(* IEC 61131-3 sources: POMIRTS_lab3/AS/Library/DPMaster, 3 files *)

(* ---- DPMaster.typ ---- *)
(********************************************************************
 * COPYRIGHT -- Bernecker + Rainer
 ********************************************************************
 * Library: DPMaster
 * File: DPMaster.typ
 * Author: B+R
 ********************************************************************
 * Data types of library DPMaster
 ********************************************************************)

TYPE
	DPDevice_typ : STRUCT			(*internal use*)
		DevType	: USINT ;
		MemorySize	: USINT ;
		DevAdress	: UDINT ;
		DevInfo	: UDINT ;
		DPIdent	: UDINT ;
		DevNumber	: UINT ;
		ConfMsgNr	: USINT ;
		CommandMsgNr	: USINT ;
		StatusMsgNr	: USINT ;
		OtherMsgNr	: USINT ;
	END_STRUCT;
END_TYPE

(* ---- DPMaster.fun ---- *)
(********************************************************************
 * COPYRIGHT -- Bernecker + Rainer
 ********************************************************************
 * Library: DPMaster
 * File: DPMaster.fun
 * Author: B+R
 ********************************************************************
 * Functions and function blocks of library DPMaster
 ********************************************************************)

FUNCTION_BLOCK DPMInit                 (*searches and initializes the specified device*)
	VAR_INPUT
		enable	:BOOL;                 (*enables execution*)
		Device	:UDINT;                (*device name given as pointer, e.g., "SL2.SS1.IF1"*)
	END_VAR
	VAR_OUTPUT
		status	:UINT;                 (*execution status: ERR_OK, ERR_FUB_ENABLE_FALSE, 0xXXXX = see help*)
		MemSize	:USINT;                (*indicates the DPM size on the card.*)
		DevIdent	:UDINT;            (*device identifier*)
		Run	:BOOL;                     (*device in run: TRUE = in run, FALSE = not in run*)
		Configuration	:BOOL;         (*configuration: TRUE = valid, FALSE = not valid*)
	END_VAR
END_FUNCTION_BLOCK

FUNCTION_BLOCK DPMio                   (*copies the input and output data areas between the B&R card and the specified buffers; asynchronous execution*)
	VAR_INPUT
		enable	:BOOL;                 (*enables execution*)
		DevIdent	:UDINT;            (*device identifier returned from DPMInit*)
		OutBuffer	:UDINT;            (*pointer to the output data area*)
		OutLen	:UDINT;                (*length of the output data area*)
		InBuffer	:UDINT;            (*pointer to the input data area*)
		InLen	:UDINT;                (*length of the input data area*)
	END_VAR
	VAR_OUTPUT
		status	:UINT;                 (*execution status: ERR_OK, ERR_FUB_ENABLE_FALSE, ERR_FUB_BUSY, 0xXXXX = see help*)
	END_VAR
	VAR
		hmode	:USINT;                (*internal variable*)
	END_VAR
END_FUNCTION_BLOCK

FUNCTION_BLOCK DPMStop                 (*stops the I/O exchange process*)
	VAR_INPUT
		enable	:BOOL;                 (*enables execution*)
		DevIdent	:UDINT;            (*device identifier returned from DPMInit*)
	END_VAR
	VAR_OUTPUT
		status	:UINT;                 (*execution status: ERR_OK, ERR_FUB_ENABLE_FALSE, 0xXXXX = see help*)
	END_VAR
END_FUNCTION_BLOCK

FUNCTION_BLOCK DPMCommand              (*Sends commands directly to bus stations; asynchronous execution*)
	VAR_INPUT
		enable	:BOOL;                 (*enables execution*)
		DevIdent	:UDINT;            (*device identifier returned from DPMInit*)
		RemoteAdress	:USINT;        (*remote slave node number, 1..126 = slave with specified node number, 127 = broadcast to all slaves*)
		GroupSelect	:USINT;            (*selects the slave group, 0 = only remoteAdress applies, 1..255 = slaves in specified goup*)
		Command	:USINT;                (*spezifies the type of command, e.g., freeze*)
	END_VAR
	VAR_OUTPUT
		status	:UINT;                 (*execution status: ERR_OK, ERR_FUB_ENABLE_FALSE, ERR_FUB_BUSY, 0xXXXX = see help*)
	END_VAR
	VAR
		istate	:UDINT;                (*internal variable*)
		waitCnt	:UINT;                 (*internal variable*)
		MessageHeader1	:USINT;        (*internal variable*)
		MessageHeader2	:USINT;        (*internal variable*)
		MessageHeader3	:USINT;        (*internal variable*)
		MessageHeader4	:USINT;        (*internal variable*)
		MessageHeader5	:USINT;        (*internal variable*)
		MessageHeader6	:USINT;        (*internal variable*)
		MessageHeader7	:USINT;        (*internal variable*)
		MessageHeader8	:USINT;        (*internal variable*)
	END_VAR
END_FUNCTION_BLOCK

FUNCTION_BLOCK DPMConfig               (*downloads the configuration; asynchronous execution*)
	VAR_INPUT
		enable	:BOOL;                 (*enables execution*)
		DevIdent	:UDINT;            (*device identifier returned from DPMInit*)
		ConfModulName	:UDINT;        (*configuration module name given as pointer*)
		Mode	:BOOL;                 (*download mode, TRUE = sequential, FALSE = in one step*)
	END_VAR
	VAR_OUTPUT
		status	:UINT;                 (*execution status: ERR_OK, ERR_FUB_ENABLE_FALSE, ERR_FUB_BUSY, 0xXXXX = see help*)
		Remaining	:UDINT;            (*displays the remaining segments until the configuration is completely loaded*)
	END_VAR
	VAR
		istate	:UDINT;                (*internal variable*)
		FileLength	:UINT;             (*internal variable*)
		waitCnt	:UINT;                 (*internal variable*)
		OffsetCopy	:UDINT;            (*internal variable*)
		pData	:UDINT;                (*internal variable*)
		Ready	:USINT;                (*internal variable*)
		FirstMessage	:BOOL;         (*internal variable*)
		MsgPutReady	:BOOL;             (*internal variable*)
	END_VAR
END_FUNCTION_BLOCK

FUNCTION_BLOCK DPMSlaveStat            (*returns the current slave status*)
	VAR_INPUT
		enable	:BOOL;                 (*enables execution*)
		DevIdent	:UDINT;            (*device identifier returned from DPMInit*)
		SlaveReady	:UDINT;            (*pointer to a 16 byte array indicating whether a slave is in data transfer mode*)
		SlaveDiag	:UDINT;            (*pointer to a 16 byte array indicating availability of diagnose information on slaves*)
	END_VAR
	VAR_OUTPUT
		status	:UINT;                 (*execution status: ERR_OK, ERR_FUB_ENABLE_FALSE, 0xXXXX = see help*)
		SlaveStatus	:BOOL;             (*TRUE = a configured slave is not in data transfer mode or has diagnostic messages*)
	END_VAR
END_FUNCTION_BLOCK

FUNCTION_BLOCK DPMSlaveExtStat         (*returns the exact status of a slave; asynchronous execution*)
	VAR_INPUT
		enable	:BOOL;                 (*enables execution*)
		DevIdent	:UDINT;            (*device identifier returned from DPMInit*)
		SlaveNumber	:USINT;            (*slave number*)
		SlaveDiagnostic	:UDINT;        (*pointer to an array of 48 bytes containing extended status and diagnostic information*)
	END_VAR
	VAR_OUTPUT
		status	:UINT;                 (*execution status: ERR_OK, ERR_FUB_ENABLE_FALSE, ERR_FUB_BUSY, 0xXXXX = see help*)
		SlaveReady	:BOOL;             (*TRUE = slave is not in data transfer mode*)
		SlaveDiag	:BOOL;             (*TRUE = slave is in diagnostics mode*)
	END_VAR
	VAR
		istate	:UDINT;               (*internal variable*)
		waitCnt	:UINT;                (*internal variable*)
	END_VAR
END_FUNCTION_BLOCK

FUNCTION_BLOCK DPMOff                  (*stops a ProfiBus DP master layer 2 communication*)
	VAR_INPUT
		enable	:BOOL;                 (*enables execution*)
		DevIdent	:UDINT;            (*device identifier returned from DPMInit*)
	END_VAR
	VAR_OUTPUT
		status	:UINT;                 (*execution status: ERR_OK, ERR_FUB_ENABLE_FALSE, 0xXXXX = see help*)
	END_VAR
END_FUNCTION_BLOCK

FUNCTION_BLOCK DPMOn                   (*starts a ProfiBus DP master layer 2 communication*)
	VAR_INPUT
		enable	:BOOL;                 (*enables execution*)
		DevIdent	:UDINT;            (*device identifier returned from DPMInit*)
	END_VAR
	VAR_OUTPUT
		status	:UINT;                 (*execution status: ERR_OK, ERR_FUB_ENABLE_FALSE, 0xXXXX = see help*)
	END_VAR
END_FUNCTION_BLOCK

FUNCTION_BLOCK DPMStart                (*starts the I/O exchange process*)
	VAR_INPUT
		enable	:BOOL;                 (*enables execution*)
		DevIdent	:UDINT;            (*device identifier returned from DPMInit*)
	END_VAR
	VAR_OUTPUT
		status	:UINT;                 (*execution status: ERR_OK, ERR_FUB_ENABLE_FALSE, 0xXXXX = see help*)
	END_VAR
END_FUNCTION_BLOCK

FUNCTION DPMSearchDevices : UINT       (*searches the target system for B&R fieldbus cards*)
	VAR_INPUT
		pInfos	:UDINT;                (*pointer to the device information structure*)
		count	:USINT;                (*number of devices to be searched*)
	END_VAR
END_FUNCTION

FUNCTION_BLOCK DPMDialog               (*send messages to the B&R card; asynchronous execution*)
	VAR_INPUT
		enable	:BOOL;                 (*enables execution*)
		DevIdent	:UDINT;            (*device identifier returned from DPMInit*)
		Message	:UDINT;                (*pointer to the message structure*)
	END_VAR
	VAR_OUTPUT
		status	:UINT;                 (*execution status: ERR_OK, ERR_FUB_ENABLE_FALSE, ERR_FUB_BUSY, 0xXXXX = see help*)
	END_VAR
	VAR
		istate	:UDINT;                (*internal variable*)
		tx	:USINT;                    (*internal variable*)
		waitCount	:UINT;             (*internal variable*)
	END_VAR
END_FUNCTION_BLOCK

FUNCTION_BLOCK DPMGetMessage           (*sends a message to the B&R card and does not wait for an answer; asynchronous execution*)
	VAR_INPUT
		enable	:BOOL;                 (*enables execution*)
		DevIdent	:UDINT;            (*device identifier returned from DPMInit*)
		Message	:UDINT;                (*pointer to the message structure*)
	END_VAR
	VAR_OUTPUT
		status	:UINT;                 (*execution status: ERR_OK, ERR_FUB_ENABLE_FALSE, ERR_FUB_BUSY, 0xXXXX = see help*)
	END_VAR
	VAR
		waitCount	:UINT;             (*internal variable*)
	END_VAR
END_FUNCTION_BLOCK

FUNCTION_BLOCK DPMPutMessage            (*reads out a message from the B&R card; asynchronous execution*)
	VAR_INPUT
		enable	:BOOL;                 (*enables execution*)
		DevIdent	:UDINT;            (*device identifier returned from DPMInit*)
		Message	:UDINT;                (*pointer to the message structure*)
	END_VAR
	VAR_OUTPUT
		status	:UINT;                 (*execution status: ERR_OK, ERR_FUB_ENABLE_FALSE, ERR_FUB_BUSY, 0xXXXX = see help*)
	END_VAR
	VAR
		waitCount	:UINT;             (*internal variable*)
	END_VAR
END_FUNCTION_BLOCK

(* ---- DPMaster.var ---- *)
(********************************************************************
 * COPYRIGHT -- Bernecker + Rainer
 ********************************************************************
 * Library: DPMaster
 * File: DPMaster.var
 * Author: B+R
 ********************************************************************
 * Local variables of library DPMaster
 ********************************************************************)

VAR CONSTANT
	ERR_USR_MASTER_IS_STOPPED	: UINT	:= 12190;		(*master not in "RUN" state*)
	ERR_USR_WRONG_HANDSHAKE	: UINT	:= 12191;		(*not supported handshake mode*)
	ERR_USR_OUTLEN_TOO_LONG	: UINT	:= 12193;		(*cannot copy so much output data*)
	ERR_USR_WRONG_DEVIDENT	: UINT	:= 12183;		(*invalid device identifier*)
	ERR_USR_INLEN_TOO_LONG	: UINT	:= 12192;		(*cannot copy so much input data*)
	ERR_USR_WRONG_MEMSIZE	: UINT	:= 12186;		(*specified memory size does not match device memory size*)
	ERR_USR_DEV_MBOX_FULL	: UINT	:= 12180;		(*mailbox full*)
	ERR_USR_WRONG_MODENR	: UINT	:= 12187;		(*specified mode number does not exist*)
	ERR_USR_NOFREEIDENT	: UINT	:= 12185;		(*no more identifier numbers available for this device*)
	host_reserved_flag	: USINT	:= 16;		(*internal constant*)
	ERR_USR_SLAVE_CONF	: UINT	:= 12189;		(*specified slave not configured*)
	ERR_USR_INTERNAL	: UINT	:= 12181;		(*internal error*)
	ERR_USR_DATA_LNG	: UINT	:= 12188;		(*incorrect data length of configuration module*)
	ERR_USR_BADIDENT	: UINT	:= 12184;		(*incorrect identifier number*)
	ERR_USR_NOIDENT	: UINT	:= 12182;		(*no identifier number for the device*)
	STATEACK_FLAG	: USINT	:= 8;		(*internal constant*)
	NOTREADY_FLAG	: USINT	:= 32;		(*internal constant*)
	MAX_DP_BOARDS	: USINT	:= 8;		(*internal constant*)
	HOSTACK_FLAG	: USINT	:= 1;		(*internal constant*)
	DEVCOM_FLAG	: USINT	:= 2;		(*internal constant*)
	RESET_FLAG	: USINT	:= 128;		(*internal constant*)
	PDCOM_FLAG	: USINT	:= 4;		(*internal constant*)
	INIT_FLAG	: USINT	:= 64;		(*internal constant*)
	WORKING	: UINT	:= 65535;		(*function block still working*)
END_VAR
